(* CODESYS project tcsups_cx51x0.library
   Company: Evolution
   Title: TcSUPS_CX51x0
   Author: Itzko Christow
   Version: 1.0.0.0

Project tree, tasks and I/O mapping:
  libraries: Tc2_Standard, * (Beckhoff Automation GmbH); Tc2_System, * (Beckhoff Automation GmbH); Tc2_Utilities, * (Beckhoff Automation GmbH)
  Data types/
    SeCO_Nds UPS/
      data type E_S_UPS_Mode
      data type E_S_UPS_State
  Global Variables/
    global variables Global_Variables
  POUs/
    SeCO_Nds UPS/
      Internal/
        function block FB_NT_QuickShutdown [ST]
      function block FB_S_UPS_CX51x0 [ST]
    function F_GetVersionTcSUPS_CX51x0 [ST]
  Visualizations/
*)

// Data types/SeCO_Nds UPS/E_S_UPS_Mode
TYPE E_S_UPS_Mode : (
	eSUPS_WrPersistData_Shutdown,			(* in case of powerfailure: writing of persistent data + shutdown*)
	eSUPS_WrPersistData_NoShutdown,			(* in case of powerfailure: writing of persistent data, no shutdown*)
	eSUPS_ImmediateShutdown,				(* in case of powerfailure: skips writing of data, immediate shutdown*)
	eSUPS_CheckPowerStatus					(* in case of powerfailure: reports powerfailure without action (no writing, no shutdown) *)
);
END_TYPE

// Data types/SeCO_Nds UPS/E_S_UPS_State
TYPE E_S_UPS_State : (
	eSUPS_PowerOK,
	eSUPS_PowerFailure,
	eSUPS_WritePersistentData,
	eSUPS_QuickShutdown,
	eSUPS_WaitForRecover,
	eSUPS_WaitForPowerOFF
);


END_TYPE

// Global Variables/Global_Variables
{attribute 'Tc2GvlVarNames'}
VAR_GLOBAL
	eGlobalSUpsState	: E_S_UPS_State; (* current ups state of S-UPS *)
END_VAR

// POUs/F_GetVersionTcSUPS_CX51x0
FUNCTION F_GetVersionTcSUPS_CX51x0 : UINT	(* Gets the library version info *)
VAR_INPUT
	nVersionElement		:	INT;
(*
	Possible nVersionElement parameter:
	1	:	major number
	2	:	minor number
	3	:	revision number
*)
END_VAR
(* Version history:
Date		|	Version			|	created with					|	Author				|	Remark
dd.mm.yyyy	|					|									|						|
-----------------------------------------------------------------------------------------------------------------------------------------------------------------------------------------------------------------------------------------------------------------------------------
12.04.2014	|	1.0.0			|	TCAT2.11 R3 B2246				|	I.Ch.				|	first release (created from TcSUPS v1.0.2)

*)

CASE nVersionElement OF
1:	(* major number *)
	F_GetVersionTcSUPS_CX51x0 := 1;
2:	(* minor number *)
	F_GetVersionTcSUPS_CX51x0 := 0;
3:	(* revision number *)
	F_GetVersionTcSUPS_CX51x0 := 0;
ELSE
	F_GetVersionTcSUPS_CX51x0 := 16#FFFF;
END_CASE

END_FUNCTION

// POUs/SeCO_Nds UPS/Internal/FB_NT_QuickShutdown
FUNCTION_BLOCK FB_NT_QuickShutdown
VAR_INPUT
	NETID				:T_AmsNetId;
	START				:BOOL;
	TMOUT				:TIME := DEFAULT_ADS_TIMEOUT;
END_VAR
VAR_OUTPUT
	BUSY				:BOOL;
	ERR					:BOOL;
	ERRID				:UDINT;
END_VAR
{library private}
VAR
	ADSWRTCTL1			:ADSWRTCTL;
	RisingEdge			:R_TRIG;
	DELAY				:DWORD := 16#FFFFFFFF;
END_VAR

RisingEdge(CLK:=START);

IF RisingEdge.Q THEN
	ADSWRTCTL1(	NETID := NETID,
					PORT := AMSPORT_R3_SYSSERV,
					ADSSTATE := ADSSTATE_POWERFAILURE,
					DEVSTATE := 0,
					LEN := SIZEOF(DELAY),
					SRCADDR :=ADR(DELAY),
					Write := TRUE,
					TMOUT := TMOUT
				);
ELSE
	ADSWRTCTL1( Write:=FALSE);
END_IF


BUSY := ADSWRTCTL1.BUSY;
ERR := ADSWRTCTL1.ERR;
ERRID := ADSWRTCTL1.ERRID;

END_FUNCTION_BLOCK

// POUs/SeCO_Nds UPS/FB_S_UPS_CX51x0
FUNCTION_BLOCK FB_S_UPS_CX51x0
VAR_INPUT
	sNetID					: T_AmsNetId 		:= ''; 								(* '' = local netid *)
	iPLCPort				: UINT 				:= AMSPORT_R0_PLC_RTS1;				(* PLC Runtime System for writing persistent data *)
	iUPSPort				: UINT 				:= 16#588;							(* Port for reading Power State of UPS, dafault 16#588 *)
	tTimeout				: TIME 				:= DEFAULT_ADS_TIMEOUT;				(* ADS Timeout *)
	eUpsMode				: E_S_UPS_Mode		:= eSUPS_WrPersistData_Shutdown;	(* UPS mode (w/wo writing persistent data, w/wo shutdown) *)
	ePersistentMode			: E_PersistentMode	:= SPDM_2PASS;						(* mode for writing persistent data *)
	tRecoverTime			: TIME 				:= T#10s;							(* ON time to recover from short power failure in mode eSUPS_WrPersistData_NoShutdown/eSUPS_CheckPowerStatus  *)
END_VAR
VAR_OUTPUT
	bPowerFailDetect		: BOOL;													(* TRUE while powerfailure is detected *)
	eState					: E_S_UPS_State;										(* current ups state *)
END_VAR
{library private}
VAR
	fbWritePersistentData	: FB_WritePersistentData;
	fbNT_QuickShutdown 		: FB_NT_QuickShutdown;
	dwTemp					: DWORD;
	WaitForOffTimer			: TON;
	bFirstCycle				: BOOL := TRUE;
	bPowerOKInFirstCycle	: BOOL := FALSE;
END_VAR

(* monitor power state *)
dwTemp := FW_PortRead(iUPSPort, NoOfByte_DWord);
bPowerFailDetect := dwTemp.22;

(* load check *)
IF bFirstCycle THEN
	bFirstCycle 			:= FALSE;
	bPowerOKInFirstCycle 	:= NOT bPowerFailDetect;
END_IF

(* UPS State Machine *)
CASE eState OF
eSUPS_PowerOK:
	IF bPowerFailDetect THEN
		eState := eSUPS_PowerFailure; 		(* report powerfailure *)
		WaitForOffTimer(IN := FALSE, PT := tRecoverTime);
	END_IF


eSUPS_PowerFailure:
	IF bPowerOKInFirstCycle THEN
		(* allow saving/shutdown because S-UPS is fully loaded *)
		CASE eUpsMode OF
		eSUPS_WrPersistData_Shutdown,			(* in case of powerfailure: writing of persistent data + shutdown *)
		eSUPS_WrPersistData_NoShutdown:			(* in case of powerfailure: writing of persistent data, no shutdown *)
			(* start writing of persistent data *)
			fbWritePersistentData(
				NETID	:= sNetID,
				PORT	:= iPLCPort,
				START	:= TRUE,
				TMOUT	:= tTimeout,
				MODE	:= ePersistentMode
			);
			eState := eSUPS_WritePersistentData;


		eSUPS_CheckPowerStatus:					(* in case of powerfailure: reports powerfailure without action (no writing, no shutdown) *)
			(* check if power recovers *)
			eState := eSUPS_WaitForRecover;


		eSUPS_ImmediateShutdown:				(* in case of powerfailure: skips writing of data, immediate shutdown *)
			(* start quick shutdown *)
			fbNT_QuickShutdown(
				NETID := sNetID,
				START := TRUE,
				TMOUT := tTimeout
			);
			eState := eSUPS_QuickShutdown;

		END_CASE
	ELSE
		(* don't allow saving/shutdown because S-UPS was not fully loaded, wait for OFF or recover *)
		eState := eSUPS_WaitForRecover;
	END_IF

eSUPS_WritePersistentData:
	(* writing of persistent data *)
	fbWritePersistentData(START	:= FALSE);

	IF eUpsMode = eSUPS_WrPersistData_NoShutdown THEN
		IF NOT fbWritePersistentData.BUSY THEN
			fbWritePersistentData(START	:= FALSE);

			(* wait for OFF *)
			eState := eSUPS_WaitForRecover;
			WaitForOffTimer(IN := FALSE, PT := tRecoverTime);
		END_IF
	ELSE
		IF NOT fbWritePersistentData.BUSY THEN
			fbWritePersistentData(START	:= FALSE);

			(* start quick shutdown *)
			fbNT_QuickShutdown(
				NETID := sNetID,
				START := TRUE,
				TMOUT := tTimeout
			);
			eState := eSUPS_QuickShutdown;
		END_IF
	END_IF


eSUPS_WaitForRecover:
	WaitForOffTimer(IN := (NOT bPowerFailDetect));
	IF WaitForOffTimer.Q THEN
		bPowerOKInFirstCycle := TRUE;
		eState := eSUPS_PowerOK; 		(* report powerOK *)
	END_IF


eSUPS_QuickShutdown:
	(* quick shutdown *)
	fbNT_QuickShutdown(START := FALSE);
	IF NOT fbNT_QuickShutdown.BUSY THEN
		fbNT_QuickShutdown(START := FALSE);

		(* wait for OFF *)
		eState := eSUPS_WaitForPowerOFF;
	END_IF


eSUPS_WaitForPowerOFF:
	(* wait for OFF *)
	eState := eSUPS_WaitForPowerOFF;

END_CASE

eGlobalSUpsState := eState;

END_FUNCTION_BLOCK
